// TIA Portal V17 export
// export: Created 2025-03-07T09:24:00.5771288Z, ExportSetting WithDefaults, DisplayName Totally Integrated Automation Portal, DisplayVersion V17 Update 8, DisplayName TIA Portal Openness, DisplayVersion V17 Update 8, DisplayName TIA Portal Version Control Interface, DisplayVersion V17, DisplayName SINAMICS Startdrive Advanced, DisplayVersion V17 SP2, DisplayName SINAMICS Startdrive G110M, G120, G120C, G120D, G120P, G115D, DisplayVersion V17 SP2, DisplayName SINAMICS Startdrive G130, G150, S120, S150, SINAMICS MV, S210, DisplayVersion V17 SP2, DisplayName STEP 7 Professional, DisplayVersion V17 Update 8, DisplayName SINUMERIK ONE STEP 7 Toolbox, DisplayVersion V17 Update 12, DisplayName SINUMERIK 840D sl STEP 7 Toolbox, DisplayVersion V17 Update 12, DisplayName STEP 7 Safety, DisplayVersion V17 Update 6, DisplayName WinCC Advanced, DisplayVersion V17 Update 8
DATA_BLOCK "DB21020_POWDER_FEEDER_1_GENERAL_UNIT_02"   // DB21020
{ DB_Accessible_From_OPC_UA := 'FALSE' }
VERSION : 0.1
// stored: AutoNumber false, DBAccessibleFromOPCUA false, DBAccessibleFromWebserver true, InstanceOfName FB21011_POWDER_FEEDER_GENERAL, InstanceOfType FB
"FB21011_POWDER_FEEDER_GENERAL"
   // VAR_INPUT
   //    iPOWDER_FEEDER_BRAKER_FAULT : Bool;
   //    iOPERATION_MODE_LINE_1 : Word;
   //    iOPERATION_MODE_LINE_2 : Word;
   //    iOPERATION_MODE_MATCHED_LINE_1 : Bool;
   //    iOPERATION_MODE_MATCHED_LINE_2 : Bool;
   //    iFEEDER_STATE_LINE_1 : Word;
   //    iFEEDER_STATE_LINE_2 : Word;
   //    iCARRIERGAS_STATUS_LINE_1 : Bool;
   //    iCARRIERGAS_STATUS_LINE_2 : Bool;
   //    iENABLED : Bool;
   // END_VAR
   // VAR_OUTPUT
   //    oCONNECT_POWDER_FEEDER : Bool;
   //    oOPERATION_MODE : Word;
   //    oPRODUCTION_MODE : Word;
   //    oSYSTEM_MODE : Word;
   //    oSTATION_IS_ALARMS : Bool;
   //    oSwitchoncondition_on : Bool;
   //    oSwitchoncondition_off : Bool;
   //    oMotion_Active_Right : Bool;
   //    oMotion_Active_Left : Bool;
   //    oLimit_right : Bool;
   //    oLimit_left : Bool;
   //    oALARM_MISMATCH_FAULT : Bool;
   //    oALARM_FEEDER_PROFINET_MODE_FAULT : Bool;
   // END_VAR
   // VAR
   //    DATA : "POWDER FEEDER GENERAL";
   //    INPUT_SETTINGS : Struct
   //       UNIT_NUMBER : Int;
   //       FEEDER_NUMBER : Int;
   //    END_STRUCT;
   // END_VAR
BEGIN
END_DATA_BLOCK
